PROGRAM MAIN
VAR

END_VAR

Read_Write_CoE();

END_PROGRAM

(* stored: Version 1.1.0.1, ProductVersion 3.1.4024.12
   POU MAIN: Id {60477fe8-29b2-43a3-80db-6bfd8fbe6435}, SpecialFunc None *)
